FUNCTION_BLOCK TEST_BYTE (* Test BYTE AND,OR,XOR *)
  (* Standard: IEC 61499-1 *)
  (* Version 0.1, 2006-09-06, JHC, Holobloc Inc, Made a SimpleFB *)
  (* Version 0.0, 2006-09-02, JHC, Holobloc Inc, Converted from TEST_BOOL. *)
  (* Compiler header: package fb.rt.test; *)
  (* Compiler classdef: SimpleFB *)
  (* Compiler Java Sun JDK 1.5.0 *)
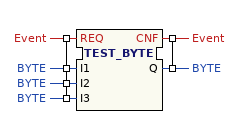
  EVENT_INPUT
    REQ WITH I1, I2, I3;
  END_EVENT
  EVENT_OUTPUT
    CNF WITH Q;
  END_EVENT
  VAR_INPUT
    I1 : BYTE;
    I2 : BYTE;
    I3 : BYTE;
  END_VAR
  VAR_OUTPUT
    Q : BYTE;
  END_VAR
  ALGORITHM REQ IN FBD:
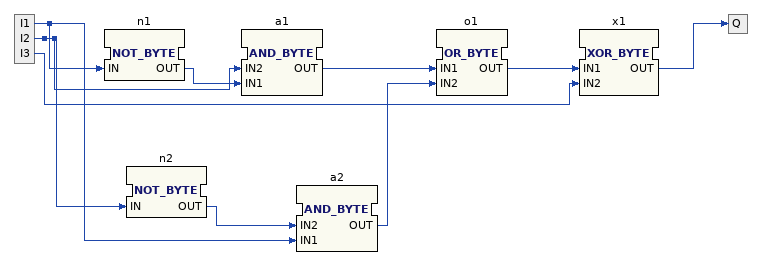
    FBS
      n1 : NOT_BYTE;
      n2 : NOT_BYTE;
      a1 : AND_BYTE;
      a2 : AND_BYTE;
      o1 : OR_BYTE;
      x1 : XOR_BYTE;
    END_FBS
    DATA_CONNECTIONS
      I1 TO n1.IN;
      I2 TO n2.IN;
      I2 TO a1.IN2;
      n2.OUT TO a2.IN2;
      n1.OUT TO a1.IN1;
      I1 TO a2.IN1;
      a1.OUT TO o1.IN1;
      a2.OUT TO o1.IN2;
      o1.OUT TO x1.IN1;
      I3 TO x1.IN2;
      x1.OUT TO Q;
    END_CONNECTIONS
  END_ALGORITHM
END_FUNCTION_BLOCK
